# EPICS autosave request: CARSApp/Db/CARS_motor_settings.req
# FILE... CARS_motor_settings.req
$(P)$(M).DHLM
$(P)$(M).DLLM
$(P)$(M).TWV
$(P)$(M).DISA
$(P)$(M).DISP
$(P)$(M).FOFF
$(P)$(M)_able.VAL
#$(P)$(M):scanParms.SP
#$(P)$(M):scanParms.EP
#$(P)$(M):scanParms.NP
